(* PLC project Untitled1, Beckhoff Automation GmbH TF6420 Database Server Query Analyser 1.0.0.0 *)
(* stored: creationDateTime 2018-12-06T16:22:40, modificationDateTime 2018-12-06T16:22:40 *)

TYPE ST_ScheduleStruct : STRUCT
  ID : LINT;
  Sequence : LINT;
  Program : LINT;
END_STRUCT;
END_TYPE
